Yaskawa INFORM job: X2_24B(90,0).JBI

/JOB
//NAME X2_24B(90,0)
///FOLDERNAME X2
//POS
///NPOS 97,97,97,6,0,0
///TOOL 0
///POSTYPE PULSE
///PULSE
C00000=-126804,-92055,-48789,-28645,51065,-65926
C00001=-154512,-17095,-20441,-46457,51312,-77671
C00002=-171755,15621,8045,-26645,28681,-67264
C00003=-172149,21602,16593,-28049,26599,-66550
C00004=-172301,24105,20177,-28733,25733,-66209
C00005=-172304,24698,22440,-29857,24778,-65655
C00006=-172303,24692,22205,-29706,24902,-65729
C00007=-172638,27660,25101,-29512,24558,-65827
C00008=-172303,24692,22205,-29706,24902,-65729
C00009=-172151,22136,18558,-28953,25772,-66100
C00010=-171757,16038,9877,-27412,27863,-66874
C00011=-172537,10567,3439,-54491,45181,-52806
C00012=-173755,15510,10864,-55609,43265,-52077
C00013=-174228,17583,13964,-56135,42495,-51750
C00014=-174231,18134,16164,-57118,41885,-51152
C00015=-174232,18056,15923,-57016,41945,-51214
C00016=-174990,20298,18026,-56800,41408,-51348
C00017=-174232,18056,15923,-57016,41945,-51214
C00018=-173759,15938,12771,-56454,42712,-51556
C00019=-172541,10889,5232,-55255,44622,-52318
C00020=-171429,14924,7459,-52899,61218,-72458
C00021=-173391,16922,12255,-53203,58903,-72125
C00022=-174169,17816,14273,-53359,57974,-71981
C00023=-174171,18372,16479,-53895,57318,-71521
C00024=-174186,18277,16037,-53778,57445,-71621
C00025=-175276,19082,16787,-53496,56785,-71865
C00026=-174186,18277,16037,-53778,57445,-71621
C00027=-173408,17346,13979,-53603,58376,-71772
C00028=-171447,15260,9091,-53255,60695,-72119
C00029=-158240,20086,12229,-60022,92490,-62238
C00030=-160039,18619,13808,-59927,90470,-61871
C00031=-160770,18111,14520,-59909,89649,-61723
C00032=-160772,18666,16726,-59889,89089,-61299
C00033=-160777,18600,16429,-59891,89163,-61359
C00034=-161819,17405,15311,-59904,88552,-61573
C00035=-160777,18600,16429,-59891,89163,-61359
C00036=-160046,19075,15684,-59897,89986,-61508
C00037=-158247,20459,14022,-59963,92011,-61877
C00038=-150109,19275,12907,-57730,110995,-56205
C00039=-150821,13979,10904,-57305,109735,-55732
C00040=-150821,14402,12600,-57021,109272,-55391
C00041=-150821,14273,12095,-57104,109409,-55492
C00042=-151158,12204,10220,-57192,109256,-55598
C00043=-150821,14043,11170,-57260,109662,-55678
C00044=-150669,18516,12396,-57787,110610,-56289
C00045=-158247,20459,14022,-59963,92011,-61877
C00046=-167890,14065,17347,-67668,61880,-42920
C00047=-169669,18211,24197,-68549,59861,-42187
C00048=-170061,18768,24798,-68558,59564,-42205
C00049=-169274,17820,25051,-68966,59844,-41773
C00050=-170061,19372,26506,-68959,59278,-41841
C00051=-170017,19530,26656,-68968,59303,-41829
C00052=-171072,19099,26318,-66111,46121,-45202
C00053=-171470,21413,27927,-59380,35158,-49884
C00054=-171439,22753,29622,-54693,28658,-52885
C00055=-171262,19099,25016,-53425,29332,-53531
C00056=-170433,12757,16140,-51044,31187,-54738
C00057=-169386,2726,-3408,-47131,59588,-64379
C00058=-162129,11944,4675,-55750,93076,-67512
C00059=-158662,2003,3434,-55371,92603,-65180
C00060=-160272,-6881,2311,-55312,89335,-64030
C00061=-159604,-3717,6096,-55247,89318,-63634
C00062=-160272,-6303,4007,-55302,88898,-63749
C00063=-167387,4235,12711,-55768,84727,-65173
C00064=-168193,4165,12704,-55860,83299,-65643
C00065=-168736,3570,12113,-55901,81787,-66173
C00066=-172154,5029,13655,-55955,75108,-68308
C00067=-176164,11624,19445,-54733,64888,-71826
C00068=-179075,18313,25454,-52030,55435,-75538
C00069=-178266,15033,21206,-51563,56009,-75939
C00070=-176209,12719,16082,-51088,58417,-76238
C00071=-169068,16735,19784,-54963,35202,-48849
C00072=-169913,23175,28896,-57292,33376,-47615
C00073=-170455,24579,30582,-57405,32871,-47577
C00074=-169641,23365,30301,-58435,33116,-46990
C00075=-170455,25081,31962,-58187,32545,-47161
C00076=-170415,25116,31996,-58212,32568,-47145
C00077=-169591,26715,33544,-58642,32829,-46891
C00078=-168079,29361,36204,-47175,23747,-53414
C00079=-167507,29848,36588,-34474,19374,-59919
C00080=-165004,30430,37169,-22964,17221,-65589
C00081=-166322,26848,32484,-19002,17862,-67498
C00082=-166314,19768,22632,-16855,20177,-68509
C00083=-168091,1601,-5375,-26856,48093,-74307
C00084=-168249,-1691,3616,-56588,64446,-69461
C00085=-170505,-28,8010,-57007,62044,-69156
C00086=-171022,1464,10464,-57260,61317,-68947
C00087=-172273,-1183,8380,-56217,57403,-70337
C00088=-172251,-1121,8431,-56221,57416,-70332
C00089=-173580,4189,12853,-54564,53300,-72010
C00090=-176732,11815,19026,-46834,42462,-77884
C00091=-178078,20393,27286,-38852,34371,-83441
C00092=-175403,21268,27072,-43793,38616,-80317
C00093=-173730,16707,19766,-43014,41026,-80711
C00094=-154512,-17095,-20441,-46457,51312,-77671
C00095=-126804,-92055,-48789,-28645,51065,-65926
C00096=2000,-92055,-48789,0,51065,0
BC00000=198883,670023,454521
BC00001=198883,753691,248108
BC00002=201955,789553,144697
BC00003=201955,789553,144697
BC00004=201955,789553,144697
BC00005=201955,789553,144697
BC00006=201955,789553,144697
BC00007=201955,789553,144697
BC00008=201955,789553,144697
BC00009=201955,789553,144697
BC00010=201955,789553,144697
BC00011=202179,789104,144548
BC00012=202179,789104,144548
BC00013=202179,789104,144548
BC00014=202179,789104,144548
BC00015=202179,789104,144548
BC00016=202179,789104,144548
BC00017=202179,789104,144548
BC00018=202179,789104,144548
BC00019=202179,789104,144548
BC00020=205866,764957,186956
BC00021=205866,764957,186956
BC00022=205866,764957,186956
BC00023=205866,764957,186956
BC00024=205866,764957,186956
BC00025=205866,764957,186956
BC00026=205866,764957,186956
BC00027=205866,764957,186956
BC00028=205866,764957,186956
BC00029=194381,744166,186587
BC00030=194381,744166,186587
BC00031=194381,744166,186587
BC00032=194381,744166,186587
BC00033=194381,744166,186587
BC00034=194381,744166,186587
BC00035=194381,744166,186587
BC00036=194381,744166,186587
BC00037=194381,744166,186587
BC00038=194381,744166,186587
BC00039=194381,744166,186587
BC00040=194381,744166,186587
BC00041=194381,744166,186587
BC00042=194381,744166,186587
BC00043=194381,744166,186587
BC00044=194381,744166,186587
BC00045=194381,744166,186587
BC00046=191404,789553,202106
BC00047=191404,789553,202106
BC00048=191404,789553,202106
BC00049=191404,789553,202106
BC00050=191404,789553,202106
BC00051=191404,789553,202106
BC00052=191404,789553,202106
BC00053=191405,789553,202103
BC00054=191405,789553,202101
BC00055=191404,789553,202106
BC00056=191404,789553,202106
BC00057=209504,770633,235142
BC00058=219057,758918,262967
BC00059=219057,758918,262967
BC00060=219057,758919,262964
BC00061=219057,758919,262964
BC00062=219057,758919,262964
BC00063=219057,758919,262964
BC00064=219057,758918,262966
BC00065=219057,758918,262966
BC00066=219057,758918,262967
BC00067=219057,758918,262967
BC00068=219057,758918,262967
BC00069=219057,758918,262967
BC00070=219057,758918,262967
BC00071=193128,789553,204744
BC00072=193128,789553,204744
BC00073=193128,789553,204744
BC00074=193128,789553,204744
BC00075=193128,789553,204744
BC00076=193128,789553,204744
BC00077=193128,789553,204744
BC00078=193128,789553,204744
BC00079=193128,789553,204744
BC00080=193128,789553,204744
BC00081=193128,789553,204744
BC00082=193128,789553,204744
BC00083=194322,770063,231438
BC00084=195310,762097,249321
BC00085=195310,762097,249321
BC00086=195310,762097,249321
BC00087=195310,762097,249321
BC00088=195310,762097,249321
BC00089=195309,762098,249319
BC00090=195309,762098,249318
BC00091=195309,762098,249318
BC00092=195310,762097,249321
BC00093=195310,762097,249321
BC00094=198883,753691,248108
BC00095=198883,670023,454521
BC00096=198883,666204,632238
EC00000=798156,0
EC00001=798156,0
EC00002=798156,0
EC00003=798156,0
EC00004=798156,0
EC00005=798156,0
EC00006=798156,0
EC00007=798156,0
EC00008=798156,0
EC00009=798156,0
EC00010=798156,0
EC00011=798156,0
EC00012=798156,0
EC00013=798156,0
EC00014=798156,0
EC00015=798156,0
EC00016=798156,0
EC00017=798156,0
EC00018=798156,0
EC00019=798156,0
EC00020=798156,0
EC00021=798156,0
EC00022=798156,0
EC00023=798156,0
EC00024=798156,0
EC00025=798156,0
EC00026=798156,0
EC00027=798156,0
EC00028=798156,0
EC00029=798156,0
EC00030=798156,0
EC00031=798156,0
EC00032=798156,0
EC00033=798156,0
EC00034=798156,0
EC00035=798156,0
EC00036=798156,0
EC00037=798156,0
EC00038=798156,0
EC00039=798156,0
EC00040=798156,0
EC00041=798156,0
EC00042=798156,0
EC00043=798156,0
EC00044=798156,0
EC00045=798156,0
EC00046=798156,0
EC00047=798156,0
EC00048=798156,0
EC00049=798156,0
EC00050=798156,0
EC00051=798156,0
EC00052=798156,0
EC00053=798155,1
EC00054=798154,1
EC00055=798156,0
EC00056=798156,0
EC00057=798156,0
EC00058=798156,0
EC00059=798156,0
EC00060=798154,1
EC00061=798154,1
EC00062=798154,1
EC00063=798154,1
EC00064=798155,0
EC00065=798155,0
EC00066=798156,0
EC00067=798156,0
EC00068=798156,0
EC00069=798156,0
EC00070=798156,0
EC00071=798156,0
EC00072=798156,0
EC00073=798156,0
EC00074=798156,0
EC00075=798156,0
EC00076=798156,0
EC00077=798156,0
EC00078=798156,0
EC00079=798156,0
EC00080=798156,0
EC00081=798156,0
EC00082=798156,0
EC00083=798156,0
EC00084=798156,0
EC00085=798156,0
EC00086=798156,0
EC00087=798156,0
EC00088=798156,0
EC00089=798156,0
EC00090=798156,0
EC00091=798156,0
EC00092=798156,0
EC00093=798156,0
EC00094=798156,0
EC00095=798156,0
EC00096=798156,0
///POSTYPE BASE
///RECTAN
///RCONF 0,0,0,0,0,0,0,0,0,0,0,0,0,0,0,0,0,0,0,0,0,0,0,0
P00006=0.222,-3.123,-1.508,0.0000,0.0000,0.0000
P00021=-0.225,-6.128,-0.405,0.0000,0.0000,0.0000
P00022=0.222,-3.123,-1.508,0.0000,0.0000,0.0000
P00023=0.143,-0.036,0.682,0.0000,0.0000,0.0000
P00024=0.145,-0.552,1.326,0.0000,0.0000,0.0000
P00030=5.926,-4.294,-1.390,0.0000,0.0000,0.0000
//INST
///DATE 2024/04/06 14:08
///ATTR SC,RW
///GROUP1 RB1,BS1
///GROUP2 ST1
NOP
'X2_24B(90,0)
MOVJ C00000 BC00000 VJ=100.00  +MOVJ EC00000 VJ=100.00
MOVJ C00001 BC00001 VJ=100.00  +MOVJ EC00001 VJ=100.00
'Path S4187
SSFTOF
SFTOF3D
MOVJ C00002 BC00002 VJ=100.00  +MOVJ EC00002 VJ=100.00
MOVL C00003 BC00003 V=800.0  +MOVJ EC00003 VJ=100.00
SMOVL C00004 BC00004 V=166.7  +MOVJ EC00004
SREFP 3 C00005 BC00005  +REFP EC00005
CALL JOB:SEARCH-R1-S13D
SET P021 P006
SFTON3D P021
SMOVL C00006 BC00006 V=166.7  +MOVJ EC00006
SREFP 3 C00007 BC00007  +REFP EC00007
CALL JOB:SEARCH-R1-S13D
SET P021 P006
SMOVL C00008 BC00008 V=166.7  +MOVJ EC00008
MOVL C00009 BC00009 V=800.0  +MOVJ EC00009 VJ=100.00
MOVL C00010 BC00010 V=1000.0  +MOVJ EC00010 VJ=100.00
'EndPath S4187
'Path S4188
SFTOF3D
MOVJ C00011 BC00011 VJ=100.00  +MOVJ EC00011 VJ=100.00
MOVL C00012 BC00012 V=800.0  +MOVJ EC00012 VJ=100.00
SMOVL C00013 BC00013 V=166.7  +MOVJ EC00013
SREFP 3 C00014 BC00014  +REFP EC00014
CALL JOB:SEARCH-R1-S13D
SET P022 P006
SFTON3D P022
SMOVL C00015 BC00015 V=166.7  +MOVJ EC00015
SREFP 3 C00016 BC00016  +REFP EC00016
CALL JOB:SEARCH-R1-S13D
SET P022 P006
SMOVL C00017 BC00017 V=166.7  +MOVJ EC00017
MOVL C00018 BC00018 V=800.0  +MOVJ EC00018 VJ=100.00
MOVL C00019 BC00019 V=1000.0  +MOVJ EC00019 VJ=100.00
'EndPath S4188
'Path S4189
SFTOF3D
MOVJ C00020 BC00020 VJ=100.00  +MOVJ EC00020 VJ=100.00
MOVL C00021 BC00021 V=800.0  +MOVJ EC00021 VJ=100.00
SMOVL C00022 BC00022 V=166.7  +MOVJ EC00022
SREFP 3 C00023 BC00023  +REFP EC00023
CALL JOB:SEARCH-R1-S13D
SET P023 P006
SFTON3D P023
SMOVL C00024 BC00024 V=166.7  +MOVJ EC00024
SREFP 3 C00025 BC00025  +REFP EC00025
CALL JOB:SEARCH-R1-S13D
SET P023 P006
SMOVL C00026 BC00026 V=166.7  +MOVJ EC00026
MOVL C00027 BC00027 V=800.0  +MOVJ EC00027 VJ=100.00
MOVL C00028 BC00028 V=1000.0  +MOVJ EC00028 VJ=100.00
'EndPath S4189
'Path S4190
SFTOF3D
MOVJ C00029 BC00029 VJ=100.00  +MOVJ EC00029 VJ=100.00
MOVL C00030 BC00030 V=800.0  +MOVJ EC00030 VJ=100.00
SMOVL C00031 BC00031 V=166.7  +MOVJ EC00031
SREFP 3 C00032 BC00032  +REFP EC00032
CALL JOB:SEARCH-R1-S13D
SET P024 P006
SFTON3D P024
SMOVL C00033 BC00033 V=166.7  +MOVJ EC00033
SREFP 3 C00034 BC00034  +REFP EC00034
CALL JOB:SEARCH-R1-S13D
SET P024 P006
SMOVL C00035 BC00035 V=166.7  +MOVJ EC00035
MOVL C00036 BC00036 V=800.0  +MOVJ EC00036 VJ=100.00
MOVL C00037 BC00037 V=1000.0  +MOVJ EC00037 VJ=100.00
'EndPath S4190
'Path W4191
SFTOF3D
SMOVL C00038 BC00038 V=1000.0  +MOVJ EC00038
SMOVL C00039 BC00039 V=166.7  +MOVJ EC00039
SREFP 3 C00040 BC00040  +REFP EC00040
CALL JOB:SEARCH-R1-S13D
SET P030 P006
SFTON3D P030
SMOVL C00041 BC00041 V=166.7  +MOVJ EC00041
SREFP 3 C00042 BC00042  +REFP EC00042
CALL JOB:SEARCH-R1-S13D
SET P030 P006
SMOVL C00043 BC00043 V=250.0  +MOVJ EC00043
SFTOF3D
MOVL C00044 BC00044 V=800.0  +MOVJ EC00044 VJ=100.00
MOVL C00045 BC00045 V=1000.0  +MOVJ EC00045 VJ=100.00
SFTON3D P022
MOVJ C00046 BC00046 VJ=100.00  +MOVJ EC00046 VJ=100.00
SMOVL C00047 BC00047 V=800.0  +MOVJ EC00047
SREFP 1 C00048 BC00048  +REFP EC00048
SREFP 2 C00049 BC00049  +REFP EC00049
SMOVL C00050 BC00050 V=166.7 PL=0  +MOVJ EC00050
MACRO1 MJ#(0) ARGF21
ARCON
SWVON WEV#(100)
SMOVC C00051 BC00051 V=9.2  +MOVJ EC00051
SMOVC C00052 BC00052 V=9.2  +MOVJ EC00052
SMOVC C00053 BC00053 V=9.2  +MOVJ EC00053
SMOVC C00054 BC00054 V=9.2  +MOVJ EC00054
ARCOF
SWVOF
SMOVL C00055 BC00055 V=800.0  +MOVJ EC00055
SMOVL C00056 BC00056 V=1000.0  +MOVJ EC00056
SFTOF3D
'EndPath W4191
MOVJ C00057 BC00057 VJ=100.00  +MOVJ EC00057 VJ=100.00
'Path W4192
SFTOF3D
SSFTOF
SFTON3D P030
MOVJ C00058 BC00058 VJ=100.00  +MOVJ EC00058 VJ=100.00
SMOVL C00059 BC00059 V=800.0  +MOVJ EC00059
SREFP 1 C00060 BC00060  +REFP EC00060
SREFP 2 C00061 BC00061  +REFP EC00061
SMOVL C00062 BC00062 V=166.7 PL=0  +MOVJ EC00062
ARCON
SWVON WEV#(100)
SMOVL C00063 BC00063 V=9.2  +MOVJ EC00063
SMOVL C00064 BC00064 V=9.2  +MOVJ EC00064
SMOVC C00065 BC00065 V=9.2  +MOVJ EC00065
SFTON3D P024
SMOVC C00066 BC00066 V=9.2  +MOVJ EC00066
SMOVC C00067 BC00067 V=9.2  +MOVJ EC00067
SMOVC C00068 BC00068 V=9.2  +MOVJ EC00068
ARCOF
SWVOF
SMOVL C00069 BC00069 V=800.0  +MOVJ EC00069
SMOVL C00070 BC00070 V=1000.0  +MOVJ EC00070
SFTOF3D
'EndPath W4192
'Path W4193
MOVJ C00071 BC00071 VJ=100.00  +MOVJ EC00071 VJ=100.00
SFTON3D P021
SMOVL C00072 BC00072 V=800.0  +MOVJ EC00072
SREFP 1 C00073 BC00073  +REFP EC00073
SREFP 2 C00074 BC00074  +REFP EC00074
SMOVL C00075 BC00075 V=166.7 PL=0  +MOVJ EC00075
ARCON
SWVON WEV#(100)
SMOVC C00076 BC00076 V=9.2  +MOVJ EC00076
SMOVC C00077 BC00077 V=9.2  +MOVJ EC00077
SMOVC C00078 BC00078 V=9.2  +MOVJ EC00078
SMOVC C00079 BC00079 V=9.2  +MOVJ EC00079
SMOVC C00080 BC00080 V=9.2  +MOVJ EC00080
ARCOF
SWVOF
SFTOF3D
SMOVL C00081 BC00081 V=800.0  +MOVJ EC00081
SMOVL C00082 BC00082 V=1000.0  +MOVJ EC00082
'EndPath W4193
MOVJ C00083 BC00083 VJ=100.00  +MOVJ EC00083 VJ=100.00
'Path W4194
MOVJ C00084 BC00084 VJ=100.00  +MOVJ EC00084 VJ=100.00
SMOVL C00085 BC00085 V=800.0  +MOVJ EC00085
SSFTOF
SFTON3D P023
SMOVL C00086 BC00086 V=166.7 PL=0  +MOVJ EC00086
ARCON
SWVON WEV#(100)
SMOVL C00087 BC00087 V=9.2  +MOVJ EC00087
SMOVC C00088 BC00088 V=9.2  +MOVJ EC00088
SMOVC C00089 BC00089 V=9.2  +MOVJ EC00089
SMOVC C00090 BC00090 V=9.2  +MOVJ EC00090
SMOVC C00091 BC00091 V=9.2  +MOVJ EC00091
ARCOF
SWVOF
SFTOF3D
SMOVL C00092 BC00092 V=800.0  +MOVJ EC00092
SMOVL C00093 BC00093 V=1000.0  +MOVJ EC00093
SSFTOF
'EndPath W4194
MOVJ C00094 BC00094 VJ=100.00  +MOVJ EC00094 VJ=100.00
MOVJ C00095 BC00095 VJ=100.00  +MOVJ EC00095 VJ=100.00
MOVJ C00096 BC00096 VJ=100.00  +MOVJ EC00096 VJ=100.00
END
